(* CODESYS project RTNNI.library
   Author: Zexu Zhou, Christoph Hinze
   Placeholder: Real-Time Neural Network generator
   Title: Real-Time Neural Network generator
   Version: 0.1
   Company: ISW

Project tree, tasks and I/O mapping:
  libraries: Tc2_Standard, * (Beckhoff Automation GmbH); Tc2_System, * (Beckhoff Automation GmbH); Tc2_Utilities, * (Beckhoff Automation GmbH); Tc3_Module, * (Beckhoff Automation GmbH)
  DUTs/
    data type act_type
    data type Layer
    data type norm_type
  GVLs/
  POUs/
    activation function/
      function F_exponential [ST]
      function F_relu [ST]
      function F_selu [ST]
      function F_sigmoid [ST]
      function F_silu [ST]
      function F_softplus [ST]
      function F_softsign [ST]
      function F_tanh [ST]
    math/
      function F_Dot [ST]
    normalization/
      function F_denormalization [ST]
      function F_normalization [ST]
      function F_NormalizationLayer [ST]
    function F_ForwardPropagation [ST]
    function block FB_LoadWeights [ST]
  VISUs/
*)

// DUTs/act_type
{attribute 'qualified_only'}
{attribute 'strict'}
TYPE act_type :
(
	linear := 0,
	relu :=1,
	tanh :=2,
	sigmoid :=3,
	softplus := 4,
	softsign := 5,
	silu := 6,
	selu := 7,
	exponential := 8
);
END_TYPE

// DUTs/Layer
TYPE Layer :
STRUCT
	num_neurons : UINT;
	activation : act_type;
	pointer_weight: POINTER TO LREAL;
	pointer_bias: POINTER TO LREAL;
	normalization: norm_type;
END_STRUCT
END_TYPE

// DUTs/norm_type
{attribute 'qualified_only'}
{attribute 'strict'}
TYPE norm_type :
(	
	none := 0,	
	normalization := 1,
	denormalization :=2
);
END_TYPE

// POUs/activation function/F_exponential
FUNCTION F_exponential : lreal
VAR_INPUT
	x : LREAL;
END_VAR

F_exponential := exp(x);

END_FUNCTION

// POUs/activation function/F_relu
FUNCTION F_relu : LREAL
VAR_INPUT
	x : LREAL;
END_VAR

IF x<0 THEN
	F_relu := 0;
ELSE
	F_relu := x;	
END_IF

END_FUNCTION

// POUs/activation function/F_selu
FUNCTION F_selu : lreal
VAR_INPUT
	x : LREAL;
END_VAR
VAR
	scale : LREAL := 1.05070098;
	alpha : LREAL := 1.67326324;
END_VAR

IF x > 0 THEN
	F_selu := scale * x;
ELSIF x < -1E2 THEN
	F_selu := - scale * alpha;
ELSE
	F_selu := scale * alpha * (exp(x) - 1);
END_IF

END_FUNCTION

// POUs/activation function/F_sigmoid
FUNCTION F_sigmoid : LREAL
VAR_INPUT
	x : LREAL;
END_VAR

IF x > 1E2 THEN
	F_sigmoid := 1;
ELSIF x < -1E2 THEN
	F_sigmoid := 0;
ELSE
	F_sigmoid := 1 / (1 + EXP(-x));
END_IF

END_FUNCTION

// POUs/activation function/F_silu
FUNCTION F_silu : lreal
VAR_INPUT
	x : LREAL;
END_VAR

IF x > 1E2 THEN
	F_silu := x;
ELSIF x < -1E2 THEN
	F_silu := 0;
ELSE
	F_silu := x / (1 + EXP(-x));
END_IF

END_FUNCTION

// POUs/activation function/F_softplus
FUNCTION F_softplus : lreal
VAR_INPUT
	x : LREAL;
END_VAR

IF x > 1E2 THEN
	F_softplus := x;
ELSIF x < -1E2 THEN
	F_softplus := 0;
ELSE
	F_softplus := LOG(EXP(x)+1);
END_IF

END_FUNCTION

// POUs/activation function/F_softsign
FUNCTION F_softsign : lreal
VAR_INPUT
	x : LREAL;
END_VAR

F_softsign := x / (abs(x) + 1);

END_FUNCTION

// POUs/activation function/F_tanh
FUNCTION F_tanh : LREAL
VAR_INPUT
	x: LREAL;
END_VAR

IF x > 1E2 THEN
	F_tanh := 1;
ELSIF x < -1E2 THEN
	F_tanh := -1;
ELSE
	F_tanh := (EXP(x) - EXP(-x))/(EXP(x) + EXP(-x));
END_IF

END_FUNCTION

// POUs/math/F_Dot
FUNCTION F_Dot : LREAL
VAR_INPUT
	vector_1: POINTER TO LREAL;
	vector_2: POINTER TO LREAL;
	length: UINT;
END_VAR
VAR
	i : UINT;
END_VAR

F_Dot := 0;
FOR i := 0 TO length-1 DO
	F_Dot := F_Dot + vector_1[i] * vector_2[i];
END_FOR

END_FUNCTION

// POUs/normalization/F_denormalization
FUNCTION F_denormalization : LREAL
VAR_INPUT
	x : LREAL;
	mean : LREAL;
	std : LREAL;
END_VAR

F_denormalization := x * std + mean;

END_FUNCTION

// POUs/normalization/F_normalization
FUNCTION F_normalization : LREAL
VAR_INPUT
	x : LREAL;
	mean : LREAL;
	std : LREAL;
END_VAR

F_normalization := (x - mean) / std;

END_FUNCTION

// POUs/normalization/F_NormalizationLayer
FUNCTION F_NormalizationLayer : BOOL
VAR_INPUT
	pointer_input : POINTER TO LREAL;
	pointer_mean : POINTER TO LREAL;
	pointer_std : POINTER TO LREAL;
	invert: BOOL;
	num_neurons : UINT;
END_VAR
VAR
	in : UINT;
	id : UINT;
END_VAR

IF NOT invert THEN
	FOR in := 0 TO num_neurons-1 DO
		pointer_input[in] := F_normalization(x:=pointer_input[in],mean:=pointer_mean[in],std:=pointer_std[in]);
	END_FOR
ELSE
	FOR id := 0 TO num_neurons-1 DO
		 pointer_input[id] := F_denormalization(x:=pointer_input[id],mean:=pointer_mean[id],std:=pointer_std[id]);
	END_FOR
END_IF

END_FUNCTION

// POUs/F_ForwardPropagation
FUNCTION F_ForwardPropagation : LREAL
VAR_INPUT
	layer_pre : Layer;
	layer_next : Layer;
	pointer_in : POINTER TO LREAL;
	pointer_out : POINTER TO LREAL; 
END_VAR
VAR
	i : UINT;
	length_in : UINT;	
	length_out : UINT;

	activation_type : act_type;
END_VAR

length_in := layer_pre.num_neurons;
length_out := layer_next.num_neurons;
activation_type := layer_next.activation;
FOR i := 0 TO length_out-1 DO
	pointer_out[i] := F_Dot(ADR(layer_next.pointer_weight[i * length_in]),pointer_in,length_in); 
	pointer_out[i] := layer_next.pointer_bias[i] + pointer_out[i];
	CASE activation_type OF
		act_type.relu:
		pointer_out[i] := F_relu(pointer_out[i]);
		act_type.tanh:
		pointer_out[i] := F_tanh(pointer_out[i]);
		act_type.exponential:
		pointer_out[i] := F_exponential(pointer_out[i]);
		act_type.selu:
		pointer_out[i] := F_selu(pointer_out[i]);
		act_type.sigmoid:
		pointer_out[i] := F_sigmoid(pointer_out[i]);
		act_type.silu:
		pointer_out[i] := F_silu(pointer_out[i]);
		act_type.softplus:
		pointer_out[i] := F_softplus(pointer_out[i]);
		act_type.softsign:
		pointer_out[i] := F_softsign(pointer_out[i]);
	ELSE
		CONTINUE;
	END_CASE
END_FOR

END_FUNCTION

// POUs/FB_LoadWeights
FUNCTION_BLOCK FB_LoadWeights
VAR_INPUT
	execute : BOOL := FALSE;
	filePath : T_MaxString;
	ReadAdr :POINTER TO LREAL;
	ReadLen : UDINT;
END_VAR
VAR_OUTPUT
	busy : BOOL ;
END_VAR
VAR
	 
	i : UINT;
	step : UINT := 1;
	fbFileOpen : FB_FileOpen;
	hFile : UINT;
	fbFileRead : FB_FileRead;
	fbFileClose : FB_FileClose;
END_VAR

CASE step OF
	1:
		busy := FALSE;
		IF execute THEN
			step := step + 1;
			busy := TRUE;
		END_IF
	2: 
		fbFileOpen(bExecute := FALSE);
		fbFileOpen(sPathName := filePath ,nMode := FOPEN_MODEREAD OR FOPEN_MODEBINARY, bExecute := TRUE);
		step := step+1;
	3:
		fbFileOpen(bExecute := FALSE);
		IF NOT fbFileOpen.bBusy THEN
			hFile := fbFileOpen.hFile;
			step := step +1;
		END_IF
	4:
		fbFileRead(bExecute := FALSE);
		fbFileRead(hFile := hFile,pReadBuff := ReadAdr ,cbReadLen := ReadLen,bEXecute := TRUE);
		step := step +1;
	5:
		fbFileRead(bExecute := FALSE);
		IF NOT fbFileRead.bBusy THEN
			fbFileClose(bExecute := FALSE);		
			fbFileClose(hFile:= hFile, bExecute := TRUE);
			step := step +1;
		END_IF
	6:
		fbFileClose(bExecute := FALSE);	
		IF NOT fbFileClose.bBusy THEN
			step := 1;
			busy := FALSE;
			execute := FALSE;
		END_IF
END_CASE

END_FUNCTION_BLOCK
